// TIA Portal V16 export
// export: Created 2023-01-03T15:35:08.2267495Z, ExportSetting WithDefaults, DisplayName Totally Integrated Automation Portal, DisplayVersion V16, DisplayName TIA Portal Version Control Interface, DisplayVersion V16, DisplayName TIA Portal Openness, DisplayVersion V16, DisplayName STEP 7 Professional, DisplayVersion V16, DisplayName STEP 7 Safety, DisplayVersion V16, DisplayName WinCC Advanced, DisplayVersion V16
DATA_BLOCK "SPEED_MOTOR"   // DB6
{ S7_Optimized_Access := 'TRUE' }
VERSION : 0.1
// stored: AutoNumber true, DBAccessibleFromOPCUA true, IsOnlyStoredInLoadMemory false, IsRetainMemResEnabled false, IsWriteProtectedInAS false, MemoryReserve 100
   VAR
      SPEED_SP { S7_SetPoint := 'True'} : Real := 14.0;
      "-B8" : Real;
      Positive_Speed : Struct
         Threshold_Error : Real := 29.0;
         Threshold_Warning : Real := 24.0;
         Error : Bool;
         Warning : Bool;
      END_STRUCT;
      Negative_Speed : Struct
         Threshold_Error : Real := -16.0;
         Threshold_Warning : Real := -14.0;
      END_STRUCT;
   END_VAR
BEGIN
END_DATA_BLOCK
